       #return_sfc21 := FILL(BVAL := #fill_value_0, BLK    =>  "CTL");
       #return_sfc21 := FILL(BVAL := #fill_value_0, BLK    =>  "CRUC");
       #return_sfc21 := FILL(BVAL := #fill_value_0, BLK    =>  "CM_SEL_CTRL_ALG_DB");
       #return_sfc21 := FILL(BVAL := #fill_value_0, BLK    =>  "AM_BY2_RP_CALC_INC_DB");
       #return_sfc21 := FILL(BVAL := #fill_value_0, BLK    =>  "AM_PRS_CTRL_DB");
       #return_sfc21 := FILL(BVAL := #fill_value_0, BLK    =>  "AM_XT_DRV_MOVE_DB");
       #return_sfc21 := FILL(BVAL := #fill_value_0, BLK    =>  "AM_CR_DRV_MOVE_DB");
       #return_sfc21 := FILL(BVAL := #fill_value_0, BLK    =>  "AM_CTRL_DB");
       #return_sfc21 := FILL(BVAL := #fill_value_0, BLK    =>  "AM_ID_DB");
       #return_sfc21 := FILL(BVAL := #fill_value_0, BLK    =>  "AM_PD_DB");
       #return_sfc21 := FILL(BVAL := #fill_value_0, BLK    =>  "AM_ME_DB");
       #return_sfc21 := FILL(BVAL := #fill_value_0, BLK    =>  "AM_DI_DB");
       #return_sfc21 := FILL(BVAL := #fill_value_0, BLK    =>  "AM_NE_DB");
       #return_sfc21 := FILL(BVAL := #fill_value_0, BLK    =>  "AM_SH_DB");
       #return_sfc21 := FILL(BVAL := #fill_value_0, BLK    =>  "AM_BY_DB");
       #return_sfc21 := FILL(BVAL := #fill_value_0, BLK    =>  "AM_EC_DB");
       #return_sfc21 := FILL(BVAL := #fill_value_0, BLK    =>  "AM_SD_DB");
       #return_sfc21 := FILL(BVAL := #fill_value_0, BLK    =>  "AM_RE_DB");
       #return_sfc21 := FILL(BVAL := #fill_value_0, BLK    =>  "AM_EMG_DB");
       #return_sfc21 := FILL(BVAL := #fill_value_0, BLK    =>  "BM_CALL_DRV_DB");
       #return_sfc21 := FILL(BVAL := #fill_value_0, BLK    =>  "BM_CALL_HTR_CTRL_DB");
       #return_sfc21 := FILL(BVAL := #fill_value_0, BLK    =>  "BM_CALL_RES_CALC_DB");
       #return_sfc21 := FILL(BVAL := #fill_value_0, BLK    =>  "BM_MCC_DB");
       //return_sfc21 := FILL_SFC21(bval := fill_value_0, blk    :=  BM_XT_WGT_CALC_DB);
       //return_sfc21 := FILL_SFC21(bval := fill_value_0, blk    :=  BM_ROT_DRV_DIR_DB);
       //return_sfc21 := FILL_SFC21(bval := fill_value_0, blk    :=  BM_OP_CALL_DB);
       //return_sfc21 := FILL_SFC21(bval := fill_value_0, blk    :=  BM_FDR_MOVE_HOME_DB);
       //return_sfc21 := FILL_SFC21(bval := fill_value_0, blk    :=  BM_FDR_SEQ_DB);
       //return_sfc21 := FILL_SFC21(bval := fill_value_0, blk    :=  BM_FDR_LEAK_TST_DB);
       #return_sfc21 := FILL(BVAL := #fill_value_0, BLK    =>  "BM_SI_FIL_REG_DB");
       //return_sfc21 := FILL_SFC21(bval := fill_value_0, blk    :=  BM_XT_ORB_DET_DB);
       #return_sfc21 := FILL(BVAL := #fill_value_0, BLK    =>  "BM_MLT_LVL_MON_DB");
       //return_sfc21 := FILL_SFC21(bval := fill_value_0, blk    :=  BM_MLT_VIB_MON_DB);
       #return_sfc21 := FILL(BVAL := #fill_value_0, BLK    =>  "BM_ACC_MAIN_DB");
END_FUNCTION

FUNCTION "CM_CYCLE_RAMP" : Void   // FC320, SCL
{ S7_Optimized_Access := 'FALSE' }
VERSION : 0.0
// --------------------------------------------------------------------------------
//     program     :    CM_CYCLE_RAMP
//     description :    ramp function, called in cycle with timeflag  
//     name        :    hp
//     date        :    04.04.2000
// 
//     revision    :    
//     name        :    
//     date        :    
// 
//                     (c)CGS
//     --------------------------------------------------------------------------------
   VAR_INPUT
      SetpVal : Real;   // setpoint
      IncVal : Real;   // increment/decrement - value
      TimeFlag : Bool;   // time control flag
      Enable : Bool;   // Ramp enable / disable
   END_VAR
   VAR_IN_OUT
      ActVal : Real;   // actual value - input/output
   END_VAR
   VAR_TEMP
      act : Real;
   END_VAR
BEGIN


   IF #Enable THEN          //** Ramp function **

       #act := #ActVal;

       IF #TimeFlag THEN                // calculation only if true

           IF #SetpVal > #act THEN
               #act := #act + #IncVal;
               IF #act > #SetpVal THEN
                   #act := #SetpVal;
               END_IF;        
           ELSE
               IF #SetpVal < #act THEN
                   #act := #act - #IncVal;
                   IF #act < #SetpVal THEN
                       #act := #SetpVal;
                   END_IF;            
               ELSE
                   #act := #SetpVal;
               END_IF;
           END_IF;

       END_IF;

       #ActVal := #act;

   ELSE                //** no ramp function **

       #ActVal := #SetpVal;

   END_IF;
END_FUNCTION

FUNCTION "PM_HAI_CONVERT" : Real   // FC400, SCL
{ S7_Optimized_Access := 'FALSE' }
VERSION : 0.0
// --------------------------------------------------------------------------------
//     program     :    PM_HAI_CONVERT
//     description :    fetch, convert and scale  analog input signal       
//     name        :    hp
//     date        :    06.09.00
// 
//     revision    :    
//     name        :    
//     date        :    
//     
// 
//                     (c)CGS
//     --------------------------------------------------------------------------------
// hardware_type  min_value    max_value    function
//      1         0            +27648       linear    (0..10 V or 0..20 mA) Siemens
//      2         -27648       +27648       linear    (+/-10 V)
//      3         0            +32766       linear    (0..10 V or 0..20 mA) Beckhoff
//      4         -32767       +32766       linear    (+/-10 V)
   VAR_INPUT
      CHANNEL : Word;
      CONVERT_PAR : Struct
         hardware_type : Int;
         convert_type : Int;
         min_value : Real;
         max_value : Real;
      END_STRUCT;
   END_VAR
   VAR_TEMP
      input_real : Real;
      max_range : Real;
      min_range : Real;
   END_VAR
BEGIN


       #input_real := INT_TO_REAL (WORD_TO_INT (#CHANNEL));               //fetch input

       IF #CONVERT_PAR.hardware_type = 1 THEN                             // ao_type 1 [0..27648/lin] 

           #max_range := 27648;                                          //input limits 
           #min_range := 0;
           IF #input_real > #max_range THEN
               #input_real := #max_range; 
           END_IF;
           IF #input_real < #min_range THEN
               #input_real := #min_range; 
           END_IF;
                                                                        //calculate input value 
           //calculate input value 
           #input_real := #input_real/#max_range;   

           //set return value
           #PM_HAI_CONVERT := #input_real;

       END_IF;


       IF #CONVERT_PAR.hardware_type = 2 THEN                             // ao_type 2 [-27648..27648/lin] 

           #max_range := 27648;                                          //input limits 
           #min_range := -27648;
           IF #input_real > #max_range THEN
               #input_real := #max_range; 
           END_IF;
           IF #input_real < #min_range THEN
               #input_real := #min_range; 
           END_IF;

           //calculate input value 
           #input_real := #input_real/#max_range;   

           //set return value
        #PM_HAI_CONVERT := #input_real;

       END_IF;


       IF #CONVERT_PAR.hardware_type = 3 THEN                         // ai_type 3 [0..32766/lin]

           #max_range := 32766;                                      //input limits 
           #min_range := 0;

           IF #input_real > #max_range THEN
               #input_real := #max_range; 
           END_IF;
           IF #input_real < #min_range THEN
               #input_real := #min_range; 
           END_IF;


           //calculate input value 
           #input_real := #input_real/#max_range; 

           //set return value
           #PM_HAI_CONVERT := #input_real;

       END_IF;


       IF #CONVERT_PAR.hardware_type = 4 THEN                  // ai_type 4 [-32767..32766/lin] 

           #max_range := 32766;                               //input limits 
           #min_range := -32767;
           IF #input_real > #max_range THEN
               #input_real := #max_range; 
           END_IF;
           IF #input_real < #min_range THEN
               #input_real := #min_range; 
           END_IF;

           //calculate input value 
           #input_real := #input_real/#max_range; 

           //set return value
           #PM_HAI_CONVERT := #input_real;

       END_IF;
END_FUNCTION

FUNCTION "PM_HAO_CONVERT" : Word   // FC401, SCL
{ S7_Optimized_Access := 'FALSE' }
VERSION : 0.0
// --------------------------------------------------------------------------------
//     program     :    PM_HAO_CONVERT
//     description :    convert, scale and write analog output signal       
//     name        :    hp
//     date        :    06.09.00
//     
//     revision    :
//     name        :
//     date        :    
//                     (c)CGS
//     --------------------------------------------------------------------------------
// hardware_type  min_value    max_value    function    
//      1         0            +27648       linear    (0..10 V or 0..20 mA)    Siemens
//      2         -27648       +27648       linear    (+/- 10 V)      
//      3         0            +32766       linear    (0..10 V or 0..20 mA)    Beckhoff
//      4         -32767       +32766       linear     (+/- 10V)
   VAR_INPUT
      OUTVALUE : Real;
      CONVERT_PAR : Struct
         hardware_type : Int;
         convert_type : Int;
         min_value : Real;
         max_value : Real;
      END_STRUCT;
   END_VAR
   VAR_TEMP
      output_real : Real;
      max_range : Real;
      min_range : Real;
   END_VAR
BEGIN


       #output_real := #OUTVALUE;                                        //fetch output value

       IF #output_real > 1.0 THEN                                          //upper input limits
           #output_real := 1.0; 
       END_IF;


       IF #CONVERT_PAR.hardware_type = 1 THEN                            // ao_type 1 [0..27648/lin] 

           IF #output_real < 0.0 THEN                                     //set lower limit
               #output_real := 0.0; 
           END_IF;

           #max_range := 27648;                                          //set output range                                  
           #min_range := 0;

           //calculate output value 
           #output_real := #output_real*#max_range;   

       END_IF;

       IF #CONVERT_PAR.hardware_type = 2 THEN                             // ao_type 2 [-27648..27648/lin] 

           IF #output_real < -1.0 THEN                                     //set lower limit
               #output_real := -1.0; 
           END_IF;

           #max_range := 27648;                                          //set output range 
           #min_range := -27648;

           //calculate output value
           #output_real := #output_real*#max_range;   

       END_IF;

       IF #CONVERT_PAR.hardware_type = 3 THEN                             // ao_type 3 [0..32766/lin] 

           IF #output_real < 0.0 THEN                                     //set lower limit
               #output_real := 0.0; 
           END_IF;

           #max_range := 32766;                                          //set output range 
           #min_range := 0;

           //calculate output value
           #output_real := #output_real*#max_range;   

       END_IF;

       IF #CONVERT_PAR.hardware_type = 4 THEN                             // ao_type 4 [-32767..32766/lin] 

           IF #output_real < -1.0 THEN                                    //set lower limit
               #output_real := -1.0; 
           END_IF;

           #max_range := 32766;                                         //set output range 
           #min_range := -32767;

           //calculate output value
           #output_real := #output_real*#max_range;   

       END_IF;

   #PM_HAO_CONVERT := INT_TO_WORD(REAL_TO_INT(#output_real));                //set return value                                           //set return value
END_FUNCTION

FUNCTION "PM_HAI" : Void   // FC402, SCL
{ S7_Optimized_Access := 'FALSE' }
VERSION : 0.0
// --------------------------------------------------------------------------------
//     program:         PM_HAI
//     description :    automatically generated PM_HAI
//     name:            hp
//     date        :    03.02.2021
// 
//     revision:
//     name:
//     Date:
//                     (c)CGS
//     --------------------------------------------------------------------------------
   VAR_TEMP
      x : Bool;
   END_VAR
BEGIN


   IF NOT "SY".SIM_ON THEN

       "HAI".TRV_ACT_POS := "PM_HAI_CONVERT" (CHANNEL := "P_HAI_TRV_ACT_POS":P, CONVERT_PAR := "CAI".CONFIG_DATA[1]);
       "HAI".TRV_ACT_POS_1 := "PM_HAI_CONVERT" (CHANNEL := "P_HAI_TRV_ACT_POS_1":P, CONVERT_PAR := "CAI".CONFIG_DATA[2]);
       "HAI".TRV_PRS_FIL_1 := "PM_HAI_CONVERT" (CHANNEL := "P_HAI_TRV_PRS_FIL_1":P, CONVERT_PAR := "CAI".CONFIG_DATA[3]);
       "HAI".TRV_PRS_FIL_2 := "PM_HAI_CONVERT" (CHANNEL := "P_HAI_TRV_PRS_FIL_2":P, CONVERT_PAR := "CAI".CONFIG_DATA[4]);
       "HAI".PYR_ACT_HTR_1_TMP := "PM_HAI_CONVERT" (CHANNEL := "P_HAI_PYR_ACT_HTR_1_TMP":P, CONVERT_PAR := "CAI".CONFIG_DATA[5]);
       "HAI".ACT_PRS_AR_VSL := "PM_HAI_CONVERT" (CHANNEL := "P_HAI_ACT_PRS_AR_VSL":P, CONVERT_PAR := "CAI".CONFIG_DATA[6]);
       "HAI".PYR_ACT_MELT_TMP := "PM_HAI_CONVERT" (CHANNEL := "P_HAI_PYR_ACT_MELT_TMP":P, CONVERT_PAR := "CAI".CONFIG_DATA[7]);
       "HAI".GCH_PCR_ACT_PRS := "PM_HAI_CONVERT" (CHANNEL := "P_HAI_GCH_PCR_ACT_PRS":P, CONVERT_PAR := "CAI".CONFIG_DATA[8]);
       "HAI".FCH_PCR_ACT_PRS := "PM_HAI_CONVERT" (CHANNEL := "P_HAI_FCH_PCR_ACT_PRS":P, CONVERT_PAR := "CAI".CONFIG_DATA[9]);
       "HAI".FCH_BAR_ACT_PRS_100 := "PM_HAI_CONVERT" (CHANNEL := "P_HAI_FCH_BAR_ACT_PRS_100":P, CONVERT_PAR := "CAI".CONFIG_DATA[10]);
       "HAI".ACC_WTR_TMP := "PM_HAI_CONVERT" (CHANNEL := "P_HAI_ACC_WTR_TMP":P, CONVERT_PAR := "CAI".CONFIG_DATA[11]);
       "HAI".ACC_WTR_PRS_IN := "PM_HAI_CONVERT" (CHANNEL := "P_HAI_ACC_WTR_PRS_IN":P, CONVERT_PAR := "CAI".CONFIG_DATA[12]);
       "HAI".ACC_WTR_FLW_OUT := "PM_HAI_CONVERT" (CHANNEL := "P_HAI_ACC_WTR_FLW_OUT":P, CONVERT_PAR := "CAI".CONFIG_DATA[13]);
       "HAI".ACC_WTR_FLW_IN := "PM_HAI_CONVERT" (CHANNEL := "P_HAI_ACC_WTR_FLW_IN":P, CONVERT_PAR := "CAI".CONFIG_DATA[14]);
       "HAI".ACC_WTR_SPL_PRS := "PM_HAI_CONVERT" (CHANNEL := "P_HAI_ACC_WTR_SPL_PRS":P, CONVERT_PAR := "CAI".CONFIG_DATA[15]);
       "HAI".ACC_SPARE_810 := "PM_HAI_CONVERT" (CHANNEL := "P_HAI_ACC_SPARE_810":P, CONVERT_PAR := "CAI".CONFIG_DATA[16]);

   END_IF;
END_FUNCTION

FUNCTION "PM_HAO" : Void   // FC403, SCL
{ S7_Optimized_Access := 'FALSE' }
VERSION : 0.0
// --------------------------------------------------------------------------------
//     program:         PM_HAO
//     description :    automatically generated PM_HAO
//     name:            hp
//     date        :    03.02.2021
// 
//     revision:
//     name:
//     Date:
//                     (c)CGS
//     --------------------------------------------------------------------------------
   VAR_TEMP
      x : Bool;
   END_VAR
BEGIN


   IF NOT "SY".SIM_ON THEN

       "P_HAO_TRV_SET_POS":P := "PM_HAO_CONVERT"(OUTVALUE := "HAO".TRV_SET_POS, CONVERT_PAR := "CAO".CONFIG_DATA[1]);
       "P_HAO_TRV_SET_POS_1":P := "PM_HAO_CONVERT"(OUTVALUE := "HAO".TRV_SET_POS_1, CONVERT_PAR := "CAO".CONFIG_DATA[2]);

   END_IF;
END_FUNCTION

FUNCTION "BM_SET_DIS_VAR" : Void   // FC503, SCL
{ S7_Optimized_Access := 'FALSE' }
VERSION : 0.0
BEGIN


       //heater 2
       //--------
       "DIS".ACT_HTR_2_AV_TMP := "AV".AVG_HTR_2_TMP;            //set display values
       "DIS".ACT_HTR_2_TMP := "AV".ACT_HTR_2_TMP;

       //pressure and gas flow
       //---------------------
       "DIS".SET_PRS_FNC   := "KYA".SET_PRS_FNC;

       "DIS".SET_GAS_1_FLW := "KYA".SET_GAS_1_FLW;
       "DIS".SET_GAS_2_FLW := "KYA".SET_GAS_2_FLW;

       "DIS".ACT_CR_POS_DIPPING    := "KYA".SET_DIP_POS_CR;
       "DIS".ACT_BDY2_LEN          := "KYA".ACT_BDY2_LEN;

       //melt contact variable copied to logging variable
       //------------------------------------------------
       "DIS".XT_MELT_CONTACT :=  INT_TO_REAL(BOOL_TO_INT("LT".XT_MELT_CONTACT));

       //Presetting after PLC restart
       //----------------------------
       IF ("SY".RUN_TIME < 5)  THEN
           "KYA".SET_XT_LFT_GN   := 1.0;     // gain values for drive calibration EKZ 2700 (old hardware)
           "KYA".SET_XT_ROT_GN   := 1.0;
           "KYA".SET_CR_LFT_GN   := 1.0;
           "KYA".SET_CR_ROT_GN   := 1.0;

           "KYA".SET_THR_CAL_FACT    := 1.0; // threshold calibration factor
       END_IF;
END_FUNCTION

ORGANIZATION_BLOCK "MAIN_OB1"   // OB1, SCL
{ S7_Optimized_Access := 'FALSE' }
VERSION : 0.0
// --------------------------------------------------------------------------------
//     program     :    MAIN_OB1
//     description :    main program scan OB1        
//     name        :    K. Kalkowski
//     date        :    01.09.99
// 
//     revision    :    AM_CALL
//     name        :    D.Bruess
//     date        :    23.11.99
//                     
//                     (c)CGS                    
//     --------------------------------------------------------------------------------
   VAR_TEMP
      OB1_EV_CLASS : Byte;   // Bits 0-3 = 1 (Coming event), Bits 4-7 = 1 (Event class 1)
      OB1_SCAN_1 : Byte;   // 1 (Cold restart scan 1 of OB 1), 3 (Scan 2-n of OB 1)
      OB1_PRIORITY : Byte;   // Priority of OB Execution
      OB1_OB_NUMBR : Byte;   // 1 (Organization block 1, OB1)
      OB1_RESERVED_1 : Byte;   // Reserved for system
      OB1_RESERVED_2 : Byte;   // Reserved for system
      OB1_PREV_CYCLE : Int;   // Cycle time of previous OB1 scan (milliseconds)
      OB1_MIN_CYCLE : Int;   // Minimum cycle time of OB1 (milliseconds)
      OB1_MAX_CYCLE : Int;   // Maximum cycle time of OB1 (milliseconds)
      OB1_DATE_TIME : Date_And_Time;   // Date and time OB1 started
   END_VAR
BEGIN

       //write cycle information
       //-----------------------
       "SY".OB1_PREV_CYCLE   :=  #OB1_PREV_CYCLE;         //Cycle time of previous OB1 scan (milliseconds)
       "SY".OB1_MIN_CYCLE    :=  #OB1_MIN_CYCLE;          //Minimum cycle time of OB1 (milliseconds)
       "SY".OB1_MAX_CYCLE    :=  #OB1_MAX_CYCLE;          //Maximum cycle time of OB1 (milliseconds)


       //call global DP diagnosis
       //------------------------
       "PM_PN_SET_FLT_MSG"();
       "CALL_PN_DIAG"();     

       //call power fail control
       //-----------------------  
      // SM_PWR_FAIL.SM_PWR_FAIL_DB();

       //ACTUAL PLC VERSION AND CONFIGURATION
       //------------------------------------
       "DIS".ACT_PLC_VERSION := "SW".ACT_PLC_VERSION;
       "DIS".ACT_PLC_CONFIG  := "SW".ACT_PLC_CONFIG;       

       //Build alarm acknowledge for one cycle
       //-------------------------------------
       "DV".ALARM_ACKN       := "KYD".ALARM_ACKN AND NOT "DV".ALARM_ACKN_OLD;
       "DV".ALARM_ACKN_OLD   := "KYD".ALARM_ACKN;

       //System Time
       //-----------
       "SysTimeFlag"();

       "PM_CALL_ST"();
       "BM_CALL"();

       //calculate crucible geometry
       // --------------------------
       "CM_CRUC_MAIN"();

       //automatic sequence
       // -----------------
       "AM_CTRL_DB"();

       //alarm management
       //----------------
       "SM_FLT_SETP_DEV_PRC_DB"();
       "SM_FLT_SET_ALM"();
       "SM_CALL_FAULT_RESET"();
END_ORGANIZATION_BLOCK

ORGANIZATION_BLOCK "ITR_1000ms_OB32"   // OB32, SCL
{ S7_Optimized_Access := 'FALSE' }
VERSION : 0.0
// --------------------------------------------------------------------------------
//     program     :    ITR_1000ms_OB32
//     description :    cyclic interrupt OB32 1000ms        
//     name        :    G. Eibelsh鋟ser
//     date        :    01.09.99
// 
//     revision    :
//     name        :
//     date        :    
//                     (c)CGS
//     --------------------------------------------------------------------------------
   VAR_TEMP
      info : Array[0..19] of Byte;
   END_VAR
BEGIN

       "SY".RUN_TIME := "SY".RUN_TIME + 1;             //count time since last reset
       "AM_TIME"();                                  //call timer function
       "BM_CALL_RES_CALC_DB"();     //calculate heater resistance
END_ORGANIZATION_BLOCK

ORGANIZATION_BLOCK "ITR_100ms_OB35"   // OB35, SCL
{ S7_Optimized_Access := 'FALSE' }
VERSION : 0.0
// --------------------------------------------------------------------------------
//     program     :    ITR_100ms_OB35
//     description :    cyclic interrupt OB35 100ms        
//     name        :    K. Kalkowski
//     date        :    01.09.99
// 
//     revision    :
//     name        :
//     date        :    
//                     (c)CGS
//     --------------------------------------------------------------------------------
   VAR_TEMP
      info : Array[0..19] of Byte;
   END_VAR
BEGIN

       "CM_CALL_100MS"();                               //call control loop modules

       IF "APC".STATUS="APC".BODY AND "APC".BYRST THEN
           "AM_BY2_RP_CALC_INC_DB"();    //call increment calc.fnc for 2nd body ramp

       END_IF;
END_ORGANIZATION_BLOCK

ORGANIZATION_BLOCK "ERR_TIME_OB80"   // OB80, SCL
{ S7_Optimized_Access := 'FALSE' }
VERSION : 0.0
// --------------------------------------------------------------------------------
//     program     :    ERR_TIME_OB80
//     description :    time error OB80        
//     name        :    K. Kalkowski
//     date        :    01.09.99
// 
//     revision    :
//     name        :
//     date        :    
//                     (c)CGS
//     --------------------------------------------------------------------------------
   VAR_TEMP
      info : Array[0..19] of Byte;
   END_VAR
BEGIN

       ;
END_ORGANIZATION_BLOCK

ORGANIZATION_BLOCK "ITR_DIAGNOSTIC_OB82"   // OB82, SCL
{ S7_Optimized_Access := 'FALSE' }
VERSION : 0.0
// --------------------------------------------------------------------------------
//     program     :    ITR_DIAGNOSTIC_OB82
//     description :    diagnostic interrupt OB82     
//     name        :    G. Eibelsh鋟ser
//     date        :    01.09.99
// 
//     revision    :
//     name        :
//     date        :    
//                     (c)CGS
//     --------------------------------------------------------------------------------
   VAR_TEMP
      info : Array[0..19] of Byte;
   END_VAR
BEGIN

    ;
END_ORGANIZATION_BLOCK

ORGANIZATION_BLOCK "ITR_MODULE_OB83"   // OB83, SCL
{ S7_Optimized_Access := 'FALSE' }
VERSION : 0.0
// --------------------------------------------------------------------------------
//     program     :    ITR_MODULE_OB83
//     description :    insert/remove module interrupt OB83 <NOT USED!>       
//     name        :    K. Kalkowski
//     date        :    01.09.99
// 
//     revision    :
//     name        :
//     date        :    
//                     (c)CGS
//     --------------------------------------------------------------------------------
   VAR_TEMP
      info : Array[0..19] of Byte;
   END_VAR
BEGIN

       ;
END_ORGANIZATION_BLOCK

ORGANIZATION_BLOCK "ERR_PRI_CLASS_OB85"   // OB85, SCL
{ S7_Optimized_Access := 'FALSE' }
VERSION : 0.0
// --------------------------------------------------------------------------------
//     program     :    ERR_PRI_CLASS_OB85
//     description :    priority class error OB85         
//     name        :    K. Kalkowski
//     date        :    01.09.99
// 
//     revision    :
//     name        :
//     date        :    
//                     (c)CGS
//     --------------------------------------------------------------------------------
   VAR_TEMP
      info : Array[0..19] of Byte;
   END_VAR
BEGIN

       ;
END_ORGANIZATION_BLOCK

ORGANIZATION_BLOCK "ERR_RACK_OB86"   // OB86, SCL
{ S7_Optimized_Access := 'FALSE' }
VERSION : 0.0
// --------------------------------------------------------------------------------
//     program     :    ERR_RACK_OB86
//     description :    rack failure OB86         
//     name        :    G. Eibelsh鋟ser
//     date        :    01.09.99
// 
//     revision    :
//     name        :
//     date        :    
//                     (c)CGS
//     --------------------------------------------------------------------------------
   VAR_TEMP
      info : Array[0..19] of Byte;
   END_VAR
BEGIN

      ;
END_ORGANIZATION_BLOCK

ORGANIZATION_BLOCK "RESET_OB100"   // OB100, SCL
{ S7_Optimized_Access := 'FALSE' }
VERSION : 0.0
// --------------------------------------------------------------------------------
//     program     :    RESET_OB100
//     description :    cold restart OB100         
//     name        :    K. Kalkowski
//     date        :    01.09.99
// 
//     revision    :
//     name        :
//     date        :    
//                     (c)CGS
//     --------------------------------------------------------------------------------
   VAR_TEMP
      info : Array[0..19] of Byte;
   END_VAR
BEGIN

       "SM_RESTART_CALL"();
   ;
END_ORGANIZATION_BLOCK

ORGANIZATION_BLOCK "ERR_PROG_OB121"   // OB121, SCL
{ S7_Optimized_Access := 'FALSE' }
VERSION : 0.0
// --------------------------------------------------------------------------------
//     program     :    ERR_PROG_OB121
//     description :    programming error OB121         
//     name        :    K. Kalkowski
//     date        :    01.09.99
// 
//     revision    :
//     name        :
//     date        :    
//                     (c)CGS
//     --------------------------------------------------------------------------------
   VAR_TEMP
      info : Array[0..19] of Byte;
   END_VAR
BEGIN

       ;
END_ORGANIZATION_BLOCK

ORGANIZATION_BLOCK "ERR_ACCESS_OB122"   // OB122, SCL
{ S7_Optimized_Access := 'FALSE' }
VERSION : 0.0
// --------------------------------------------------------------------------------
//     program     :    ERR_ACCESS_OB122
//     description :    access error OB122        
//     name        :    K. Kalkowski
//     date        :    01.09.99
// 
//     revision    :
//     name        :
//     date        :    
//                     (c)CGS
//     --------------------------------------------------------------------------------
   VAR_TEMP
      info : Array[0..19] of Byte;
   END_VAR
BEGIN

       ;
END_ORGANIZATION_BLOCK

// ===== PLC "CPU 315-2 PN/DP"  Unspecific CPU S7 300 =====
// protected blocks, not shown: "ERR_ACCESS_OB122", "ERR_PRI_CLASS_OB85", "ERR_PROG_OB121", "ERR_RACK_OB86", "ERR_TIME_OB80", "IO_LINK_MASTER", "ITR_1000ms_OB32", "ITR_100ms_OB35", "ITR_DIAGNOSTIC_OB82", "RESET_OB100"

VAR_GLOBAL   // PLC tag table "STEP7 classic symbols"
   "Tag_1" AT %ED1028 : DWord;
   "Tag_2" AT %AD256 : DWord;
   "Tag_3" AT %EB1032 : Byte;
   "Tag_4" AT %AB260 : Byte;
   "Tag_5" AT %ED1037 : DWord;
   "Tag_6" AT %AD262 : DWord;
   "Tag_7" AT %EB1041 : Byte;
   "Tag_8" AT %AB266 : Byte;
   "Tag_9" AT %ED1046 : DWord;
   "Tag_10" AT %AD268 : DWord;
   "Tag_11" AT %EB1050 : Byte;
   "Tag_12" AT %AB272 : Byte;
   "Tag_13" AT %ED1055 : DWord;
   "Tag_14" AT %AD274 : DWord;
   "Tag_15" AT %EB1059 : Byte;
   "Tag_16" AT %AB278 : Byte;
   "Tag_17" AT %ED1064 : DWord;
   "Tag_18" AT %AD280 : DWord;
   "Tag_19" AT %EB1068 : Byte;
   "Tag_20" AT %AB284 : Byte;
   "Tag_21" AT %ED1073 : DWord;
   "Tag_22" AT %AD286 : DWord;
   "Tag_23" AT %EB1077 : Byte;
   "Tag_24" AT %AB290 : Byte;
   "Tag_25" AT %ED1100 : DWord;
   "Tag_26" AT %AD304 : DWord;
   "Tag_27" AT %EB1104 : Byte;
   "Tag_28" AT %AB308 : Byte;
   "Tag_29" AT %ED1109 : DWord;
   "Tag_30" AT %AD310 : DWord;
   "Tag_31" AT %EB1113 : Byte;
   "Tag_32" AT %AB314 : Byte;
   "Tag_33" AT %ED1118 : DWord;
   "Tag_34" AT %AD316 : DWord;
   "Tag_35" AT %EB1122 : Byte;
   "Tag_36" AT %AB320 : Byte;
   "Tag_37" AT %ED1127 : DWord;
   "Tag_38" AT %AD322 : DWord;
   "Tag_39" AT %EB1131 : Byte;
   "Tag_40" AT %AB326 : Byte;
   "Tag_41" AT %ED1136 : DWord;
   "Tag_42" AT %AD328 : DWord;
   "Tag_43" AT %EB1140 : Byte;
   "Tag_44" AT %AB332 : Byte;
   "Tag_45" AT %ED1172 : DWord;
   "Tag_46" AT %AD352 : DWord;
   "Tag_47" AT %EB1176 : Byte;
   "Tag_48" AT %AB356 : Byte;
   "Tag_49" AT %ED1181 : DWord;
   "Tag_50" AT %AD358 : DWord;
   "Tag_51" AT %EB1185 : Byte;
   "Tag_52" AT %AB362 : Byte;
   "Tag_53" AT %ED1190 : DWord;
   "Tag_54" AT %AD364 : DWord;
   "Tag_55" AT %EB1194 : Byte;
   "Tag_56" AT %AB368 : Byte;
   "Tag_57" AT %ED1199 : DWord;
   "Tag_58" AT %AD370 : DWord;
   "Tag_59" AT %EB1203 : Byte;
   "Tag_60" AT %AB374 : Byte;
   "Tag_61" AT %ED1208 : DWord;
   "Tag_62" AT %AD376 : DWord;
   "Tag_63" AT %EB1212 : Byte;
   "Tag_64" AT %AB380 : Byte;
   "Tag_65" AT %ED1217 : DWord;
   "Tag_66" AT %AD382 : DWord;
   "Tag_67" AT %EB1221 : Byte;
   "Tag_68" AT %AB386 : Byte;
   "Tag_69" AT %ED1226 : DWord;
   "Tag_70" AT %AD388 : DWord;
   "Tag_71" AT %EB1230 : Byte;
   "Tag_72" AT %AB392 : Byte;
   "Tag_73" AT %ED1244 : DWord;
   "Tag_74" AT %AD400 : DWord;
   "Tag_75" AT %EB1248 : Byte;
   "Tag_76" AT %AB404 : Byte;
   "Tag_77" AT %ED1253 : DWord;
   "Tag_78" AT %AD406 : DWord;
   "Tag_79" AT %EB1257 : Byte;
   "Tag_80" AT %AB410 : Byte;
   "Tag_81" AT %ED1262 : DWord;
   "Tag_82" AT %AD412 : DWord;
   "Tag_83" AT %EB1266 : Byte;
   "Tag_84" AT %AB416 : Byte;
   "Tag_85" AT %ED1271 : DWord;
   "Tag_86" AT %AD418 : DWord;
   "Tag_87" AT %EB1275 : Byte;
   "Tag_88" AT %AB422 : Byte;
   "Tag_89" AT %ED1280 : DWord;
   "Tag_90" AT %AD424 : DWord;
   "Tag_91" AT %EB1284 : Byte;
   "Tag_92" AT %AB428 : Byte;
   "Tag_93" AT %ED1289 : DWord;
   "Tag_94" AT %AD430 : DWord;
   "Tag_95" AT %EB1293 : Byte;
   "Tag_96" AT %AB434 : Byte;
END_VAR

ORGANIZATION_BLOCK "MAIN_OB1"   // OB1, STL
TITLE = "Main Program Sweep (Cycle)"
{ S7_Optimized_Access := 'FALSE' }
VERSION : 0.1
// ifm io-link master Adresse transport
   VAR_TEMP
      OB1_EV_CLASS : Byte;   // Bits 0-3 = 1 (Coming event), Bits 4-7 = 1 (Event class 1)
      OB1_SCAN_1 : Byte;   // 1 (Cold restart scan 1 of OB 1), 3 (Scan 2-n of OB 1)
      OB1_PRIORITY : Byte;   // Priority of OB Execution
      OB1_OB_NUMBR : Byte;   // 1 (Organization block 1, OB1)
      OB1_RESERVED_1 : Byte;   // Reserved for system
      OB1_RESERVED_2 : Byte;   // Reserved for system
      OB1_PREV_CYCLE : Int;   // Cycle time of previous OB1 scan (milliseconds)
      OB1_MIN_CYCLE : Int;   // Minimum cycle time of OB1 (milliseconds)
      OB1_MAX_CYCLE : Int;   // Maximum cycle time of OB1 (milliseconds)
      OB1_DATE_TIME : Date_And_Time;   // Date and time OB1 started
   END_VAR
BEGIN

REGION Network 1

   //-------------------  crucible shaft
         L     "Tag_1":P;  // masse flow and temperature 4 Bytes transfer to I-Device
         T     "Tag_2":P;

         L     "Tag_3":P;  // PQI Status 2 Bytes transfer to I-Device
         T     "Tag_4":P;

   //-------------------- High current cable heater 1
         L     "Tag_5":P;
         T     "Tag_6":P;

         L     "Tag_7":P;
         T     "Tag_8":P;

   //-------------------- High current cable heater 2
         L     "Tag_9":P;
         T     "Tag_10":P;

         L     "Tag_11":P;
         T     "Tag_12":P;

   //-------------------- seed shaft
         L     "Tag_13":P;
         T     "Tag_14":P;

         L     "Tag_15":P;
         T     "Tag_16":P;

   //-------------------- Power supply heater
         L     "Tag_17":P;
         T     "Tag_18":P;

         L     "Tag_19":P;
         T     "Tag_20":P;

   //-------------------- gate chamber
         L     "Tag_21":P;
         T     "Tag_22":P;

         L     "Tag_23":P;
         T     "Tag_24":P;
   //-------------------- spare
   //      L     PED 1082
   //      T     PAD  292

   //      L     PEW 1086
   //      T     PAW  296

   //-------------------- spare
   //      L     PED 1091
   //      T     PAD  298

   //      L     PEW 1095
   //      T     PAW  302

   //-------------------- gate valve housing
         L     "Tag_25":P;
         T     "Tag_26":P;

         L     "Tag_27":P;
         T     "Tag_28":P;

   //-------------------- gate valve
         L     "Tag_29":P;
         T     "Tag_30":P;

         L     "Tag_31":P;
         T     "Tag_32":P;
   //-------------------- view port
         L     "Tag_33":P;
         T     "Tag_34":P;

         L     "Tag_35":P;
         T     "Tag_36":P;

   //-------------------- Gate chamber- view ports and bellow
         L     "Tag_37":P;
         T     "Tag_38":P;

         L     "Tag_39":P;
         T     "Tag_40":P;

   //-------------------- top chamber
         L     "Tag_41":P;
         T     "Tag_42":P;

         L     "Tag_43":P;
         T     "Tag_44":P;

   //-------------------- spare
   //     L     PED 1145
   //      T     PAD  334

   //      L     PEW 1149
   //      T     PAW  338

   //-------------------- spare
   //      L     PED 1154
   //      T     PAD  340

   //      L     PEW 1158
   //      T     PAW  344

   //-------------------- spare
   //      L     PED 1163
   //      T     PAD  346

   //      L     PEW 1167
   //      T     PAW  350   *)

   //-------------------- technology flange
         L     "Tag_45":P;
         T     "Tag_46":P;

         L     "Tag_47":P;
         T     "Tag_48":P;
   //-------------------- magnet compressor unit 4

         L     "Tag_49":P;
         T     "Tag_50":P;

         L     "Tag_51":P;
         T     "Tag_52":P;

   //-------------------- magnet compressor unit 3
         L     "Tag_53":P;
         T     "Tag_54":P;

         L     "Tag_55":P;
         T     "Tag_56":P;

   //-------------------- upper furnace vessel
         L     "Tag_57":P;
         T     "Tag_58":P;

         L     "Tag_59":P;
         T     "Tag_60":P;

   //-------------------- magnet compressor unit 2
         L     "Tag_61":P;
         T     "Tag_62":P;

         L     "Tag_63":P;
         T     "Tag_64":P;
   //-------------------- lower furnace vessel

         L     "Tag_65":P;
         T     "Tag_66":P;

         L     "Tag_67":P;
         T     "Tag_68":P;
   //-------------------- magnet compressor unit 1

         L     "Tag_69":P;
         T     "Tag_70":P;

         L     "Tag_71":P;
         T     "Tag_72":P;
   //-------------------- spare

   //      L     PED 1235
   //      T     PAD  394

   //      L     PEW 1239
   //      T     PAW  398

   //-------------------- bottom chamber
         L     "Tag_73":P;
         T     "Tag_74":P;

         L     "Tag_75":P;
         T     "Tag_76":P;
   //-------------------- Power supply magnet

         L     "Tag_77":P;
         T     "Tag_78":P;

         L     "Tag_79":P;
         T     "Tag_80":P;

   //-------------------- Socket bottom chamber
         L     "Tag_81":P;
         T     "Tag_82":P;

         L     "Tag_83":P;
         T     "Tag_84":P;

   //-------------------- Current feed through heater 1
         L     "Tag_85":P;
         T     "Tag_86":P;

         L     "Tag_87":P;
         T     "Tag_88":P;

   //-------------------- Current feed through heater 2
         L     "Tag_89":P;
         T     "Tag_90":P;

         L     "Tag_91":P;
         T     "Tag_92":P;

   //-------------------- vacuum bypass tube
         L     "Tag_93":P;
         T     "Tag_94":P;

         L     "Tag_95":P;
         T     "Tag_96":P;

   //-------------------- spare
   //     L     PED 1298
   //     T     PAD  436

   //     L     PEB 1302
   //     T     PAB  440

   //-------------------- spare
   //     L     PED 1307
   //     T     PAD  442

   //     L     PEB 1311
   //     T     PAB  446
END_REGION
END_ORGANIZATION_BLOCK

ORGANIZATION_BLOCK "I/O_FLT2"   // OB83, STL
TITLE = "I/O Point Fault"
{ S7_Optimized_Access := 'FALSE' }
VERSION : 0.1
   VAR_TEMP
      OB83_EV_CLASS : Byte;   // 16#38/39, Event class 3, module inserted/removed (8/9)
      OB83_FLT_ID : Byte;   // 16#XX, Fault identifcation code
      OB83_PRIORITY : Byte;   // Priority of OB Execution
      OB83_OB_NUMBR : Byte;   // 83 (Organization block 83, OB83)
      OB83_RESERVED_1 : Byte;   // Reserved for system
      OB83_MDL_ID : Byte;   // Input module (01010100), Output module (01010101)
      OB83_MDL_ADDR : Word;   // Base address of module with point fault
      OB83_RACK_NUM : Int;   // Number of rack that has module with point fault
      OB83_MDL_TYPE : Word;   // Module type with point fault
      OB83_DATE_TIME : Date_And_Time;   // Date and time OB83 started
   END_VAR
BEGIN
END_ORGANIZATION_BLOCK

// ===== PLC "Mig_PVA_AWL"  Unspecific CPU S7 300 =====
// protected blocks, not shown: "AG_LRECV_LF", "AG_LSEND_LF", "AG_RECV", "AG_SEND", "DCO_ReadDriveParameter", "DCO_WriteDriveParameter", "GLOBAL_DP_DIAG", "IO_LINK_DEVICE", "IO_LINK_MASTER"

VAR_GLOBAL   // PLC tag table "Default tag table"
   "Tag_1" AT %M0.0 : Bool;
   "Tag_2" AT %M0.1 : Bool;
   "Tag_3" AT %M1.0 : Bool;
   "Tag_4" AT %M1.1 : Bool;
   "Tag_5" AT %M1.2 : Bool;
   "Tag_6" AT %M1.3 : Bool;
   "Tag_7" AT %M1.4 : Bool;
   "Tag_8" AT %M1.5 : Bool;
   "Tag_9" AT %M1.6 : Bool;
   "Tag_10" AT %M1.7 : Bool;
   "Tag_11" AT %M2.0 : Bool;
   "Tag_12" AT %M3.0 : Bool;
   "Tag_13" AT %M3.1 : Bool;
   "Tag_14" AT %M2.1 : Bool;
   "Tag_15" AT %M3.2 : Bool;
   "Tag_16" AT %M3.3 : Bool;
   "Tag_17" AT %M2.2 : Bool;
   "Tag_18" AT %M3.4 : Bool;
   "Tag_19" AT %M3.5 : Bool;
   "Tag_20" AT %M2.3 : Bool;
   "Tag_21" AT %M3.6 : Bool;
   "Tag_22" AT %M3.7 : Bool;
   "Tag_23" AT %M2.4 : Bool;
   "Tag_24" AT %M4.0 : Bool;
   "Tag_25" AT %M4.1 : Bool;
   "Tag_26" AT %M2.5 : Bool;
   "Tag_27" AT %M4.2 : Bool;
   "Tag_28" AT %M4.3 : Bool;
   "Tag_29" AT %M2.6 : Bool;
   "Tag_30" AT %M4.4 : Bool;
   "Tag_31" AT %M4.5 : Bool;
   "Tag_32" AT %M2.7 : Bool;
   "Tag_33" AT %M4.6 : Bool;
   "Tag_34" AT %M4.7 : Bool;
END_VAR

DATA_BLOCK "BM_GRW_REC_BOOL"   // DB701
{ S7_Optimized_Access := 'FALSE' }
VERSION : 0.0
// --------------------------------------------------------------------------------
// program:             GRW_REC_BOOL
// description :        bool data for growth record
// name:                mb
// date        :        27.11.09 
// --------------------------------------------------------------------------------
   VAR
      phase_restart : Bool;   // Phase wurde neu gestartet
      phase_spare_02 : Bool;
      phase_spare_03 : Bool;
      phase_spare_04 : Bool;
      phase_spare_05 : Bool;
      phase_spare_06 : Bool;
      phase_spare_07 : Bool;
      phase_spare_08 : Bool;
      phase_spare_09 : Bool;
      phase_spare_10 : Bool;   // pump down
      pd_min_prs_reached : Bool;   // min. Druck erreicht
      pd_failed : Bool;   // Leckrate (0=ok/1=nicht ok)
      pd_new_seed : Bool;   // neuer Impfling bei Prozesstart
      pd_spare_04 : Bool;
      pd_spare_05 : Bool;
      pd_spare_06 : Bool;
      pd_spare_07 : Bool;
      pd_spare_08 : Bool;
      pd_spare_09 : Bool;
      pd_spare_10 : Bool;   // melting
      me_completed : Bool;   // Einschmelzen beendet (von Kamera erkannt)
      me_spare_02 : Bool;
      me_spare_03 : Bool;
      me_spare_04 : Bool;
      me_spare_05 : Bool;
      me_spare_06 : Bool;
      me_spare_07 : Bool;
      me_spare_08 : Bool;
      me_spare_09 : Bool;
      me_spare_10 : Bool;   // dipping
      di_new_seed : Bool;   // alter oder neuer Impfling (0=alt/1=neu)
      di_shield_dn : Bool;   // Trichter ist unten
      di_spare_03 : Bool;
      di_spare_04 : Bool;
      di_spare_05 : Bool;
      di_spare_06 : Bool;
      di_spare_07 : Bool;
      di_spare_08 : Bool;
      di_spare_09 : Bool;
      di_spare_10 : Bool;   // neck
      ne_spare_01 : Bool;
      ne_spare_02 : Bool;
      ne_spare_03 : Bool;
      ne_spare_04 : Bool;
      ne_spare_05 : Bool;
      ne_spare_06 : Bool;
      ne_spare_07 : Bool;
      ne_spare_08 : Bool;
      ne_spare_09 : Bool;
      ne_spare_10 : Bool;   // shoulder
      sh_spare_01 : Bool;
      sh_spare_02 : Bool;
      sh_spare_03 : Bool;
      sh_spare_04 : Bool;
      sh_spare_05 : Bool;
      sh_spare_06 : Bool;
      sh_spare_07 : Bool;
      sh_spare_08 : Bool;
      sh_spare_09 : Bool;
      sh_spare_10 : Bool;   // body
      by_spare_01 : Bool;
      by_spare_02 : Bool;
      by_spare_03 : Bool;
      by_spare_04 : Bool;
      by_spare_05 : Bool;
      by_spare_06 : Bool;
      by_spare_07 : Bool;
      by_spare_08 : Bool;
      by_spare_09 : Bool;
      by_spare_10 : Bool;   // endcone
      ec_spare_01 : Bool;
      ec_spare_02 : Bool;
      ec_spare_03 : Bool;
      ec_spare_04 : Bool;
      ec_spare_05 : Bool;
      ec_spare_06 : Bool;
      ec_spare_07 : Bool;
      ec_spare_08 : Bool;
      ec_spare_09 : Bool;
      ec_spare_10 : Bool;   // shut down
      sd_spare_01 : Bool;
      sd_spare_02 : Bool;
      sd_spare_03 : Bool;
      sd_spare_04 : Bool;
      sd_spare_05 : Bool;
      sd_spare_06 : Bool;
      sd_spare_07 : Bool;
      sd_spare_08 : Bool;
      sd_spare_09 : Bool;
      sd_spare_10 : Bool;   // removal
      re_active : Bool;   // Entnahme wurde ausgef黨rt
      re_spare_02 : Bool;
      re_spare_03 : Bool;
      re_spare_04 : Bool;
      re_spare_05 : Bool;
      re_spare_06 : Bool;
      re_spare_07 : Bool;
      re_spare_08 : Bool;
      re_spare_09 : Bool;
      re_spare_10 : Bool;   // melting back
      mb_spare_01 : Bool;
      mb_spare_02 : Bool;
      mb_spare_03 : Bool;
      mb_spare_04 : Bool;
      mb_spare_05 : Bool;
      mb_spare_06 : Bool;
      mb_spare_07 : Bool;
      mb_spare_08 : Bool;
      mb_spare_09 : Bool;
      mb_spare_10 : Bool;   // interne Speicherbits
      pd_sps_spare_01 : Bool;
      pd_sps_spare_02 : Bool;
      pd_sps_spare_03 : Bool;
      pd_sps_spare_04 : Bool;
      pd_sps_spare_05 : Bool;
      pd_sps_spare_06 : Bool;
      pd_sps_spare_07 : Bool;
      pd_sps_spare_08 : Bool;
      pd_sps_spare_09 : Bool;
      pd_sps_spare_10 : Bool;
      me_sps_spare_01 : Bool;
      me_sps_spare_02 : Bool;
      me_sps_spare_03 : Bool;
      me_sps_spare_04 : Bool;
      me_sps_spare_05 : Bool;
      me_sps_spare_06 : Bool;
      me_sps_spare_07 : Bool;
      me_sps_spare_08 : Bool;
      me_sps_spare_09 : Bool;
      me_sps_spare_10 : Bool;
      di_init_melt_temp : Bool;   // speichern Anfangs-Schmelzbadtemp. ausgef黨rt
      di_time_until_dip : Bool;   // speichern der Zeit bis Impfling in Schmelze ausgef黨rt
      di_sps_spare_03 : Bool;
      di_sps_spare_04 : Bool;
      di_sps_spare_05 : Bool;
      di_sps_spare_06 : Bool;
      di_sps_spare_07 : Bool;
      di_sps_spare_08 : Bool;
      di_sps_spare_09 : Bool;
      di_sps_spare_10 : Bool;
      ne_init_xt_pos : Bool;   // speichern Anfangs-Kristallpos. ausgef黨rt
      ne_init_cr_pos : Bool;   // speichern Anfangs-Tiegelposition ausgef黨rt
      ne_init_melt_temp : Bool;   // speichern Anfangs-Schmelzbadtemp. ausgef黨rt
      ne_low_temp_inc : Bool;   // speichern niedrigstes Temp.Inkrement ausgef黨rt
      ne_init_htr_temp : Bool;   // speichern Heizertemp
      ne_sps_spare_06 : Bool;
      ne_sps_spare_07 : Bool;
      ne_sps_spare_08 : Bool;
      ne_sps_spare_09 : Bool;
      ne_sps_spare_10 : Bool;
      sh_start_dia : Bool;   // speichern Startdurchmesser ausgef黨rt
      sh_init_htr_temp : Bool;   // speichern Heizertemp
      sh_sps_spare_03 : Bool;
      sh_sps_spare_04 : Bool;
      sh_sps_spare_05 : Bool;
      sh_sps_spare_06 : Bool;
      sh_sps_spare_07 : Bool;
      sh_sps_spare_08 : Bool;
      sh_sps_spare_09 : Bool;
      sh_sps_spare_10 : Bool;
      by_low_temp_inc : Bool;   // speichern niedrigstes Temp.Inkrement ausgef黨rt
      by_first_dia : Bool;   // speichern Startdurchmesser ausgef黨rt
      by_init_htr_temp : Bool;   // speichern Heizertemp
      by_sps_spare_04 : Bool;
      by_sps_spare_05 : Bool;
      by_sps_spare_06 : Bool;
      by_sps_spare_07 : Bool;
      by_sps_spare_08 : Bool;
      by_sps_spare_09 : Bool;
      by_sps_spare_10 : Bool;
      ec_init_htr_temp : Bool;   // speichern Heizertemp
      ec_sps_spare_02 : Bool;
      ec_sps_spare_03 : Bool;
      ec_sps_spare_04 : Bool;
      ec_sps_spare_05 : Bool;
      ec_sps_spare_06 : Bool;
      ec_sps_spare_07 : Bool;
      ec_sps_spare_08 : Bool;
      ec_sps_spare_09 : Bool;
      ec_sps_spare_10 : Bool;
      sd_sps_spare_01 : Bool;
      sd_sps_spare_02 : Bool;
      sd_sps_spare_03 : Bool;
      sd_sps_spare_04 : Bool;
      sd_sps_spare_05 : Bool;
      sd_sps_spare_06 : Bool;
      sd_sps_spare_07 : Bool;
      sd_sps_spare_08 : Bool;
      sd_sps_spare_09 : Bool;
      sd_sps_spare_10 : Bool;
      re_next_cr_pos : Bool;   // speichern Tiegelposition f黵 n鋍hstes Ankeimen ausgef黨rt
      re_sps_spare_02 : Bool;
      re_sps_spare_03 : Bool;
      re_sps_spare_04 : Bool;
      re_sps_spare_05 : Bool;
      re_sps_spare_06 : Bool;
      re_sps_spare_07 : Bool;
      re_sps_spare_08 : Bool;
      re_sps_spare_09 : Bool;
      re_sps_spare_10 : Bool;
      mb_sps_spare_01 : Bool;
      mb_sps_spare_02 : Bool;
      mb_sps_spare_03 : Bool;
      mb_sps_spare_04 : Bool;
      mb_sps_spare_05 : Bool;
      mb_sps_spare_06 : Bool;
      mb_sps_spare_07 : Bool;
      mb_sps_spare_08 : Bool;
      mb_sps_spare_09 : Bool;
      mb_sps_spare_10 : Bool;
   END_VAR
BEGIN
END_DATA_BLOCK

DATA_BLOCK "BM_GRW_REC_DINT"   // DB702
{ S7_Optimized_Access := 'FALSE' }
VERSION : 0.0
// --------------------------------------------------------------------------------
// program     :        GRW_REC_DINT
// description :        dint data for growth record
// name        :        mb
// date        :        27.11.09
// --------------------------------------------------------------------------------
   VAR
      elapsed_time : DInt;   // gesamte Prozesszeit
      phase_spare_02 : DInt;
      phase_spare_03 : DInt;
      phase_spare_04 : DInt;
      phase_spare_05 : DInt;
      phase_spare_06 : DInt;
      phase_spare_07 : DInt;
      phase_spare_08 : DInt;
      phase_spare_09 : DInt;
      phase_spare_10 : DInt;
      pd_elapsed_time : DInt;   // insgesamt vergangene Prozesszeit
      pd_phase_time : DInt;   // aktuelle/letzte Phasendauer
      pd_to_min_prs : DInt;   // Zeit bis Enddruck erreicht
      pd_retry : DInt;
      pd_spare_05 : DInt;
      pd_spare_06 : DInt;
      pd_spare_07 : DInt;
      pd_spare_08 : DInt;
      pd_spare_09 : DInt;
      pd_spare_10 : DInt;
      me_elapsed_time : DInt;   // insgesamt vergangene Prozesszeit
      me_phase_time : DInt;   // aktuelle/letzte Phasendauer
      me_melt_time : DInt;   // Zeit bis Aufschmelzen beendet
      me_spare_04 : DInt;
      me_spare_05 : DInt;
      me_spare_06 : DInt;
      me_spare_07 : DInt;
      me_spare_08 : DInt;
      me_spare_09 : DInt;
      me_spare_10 : DInt;
      di_elapsed_time : DInt;   // insgesamt vergangene Prozesszeit
      di_phase_time : DInt;   // aktuelle/letzte Phasendauer
      di_shield_dn : DInt;   // Zeit bis Trichter unten
      di_time_until_dip : DInt;   // Zeit bis Impfling in Schmelze
      di_spare_05 : DInt;
      di_spare_06 : DInt;
      di_spare_07 : DInt;
      di_spare_08 : DInt;
      di_spare_09 : DInt;
      di_spare_10 : DInt;
      ne_elapsed_time : DInt;   // insgesamt vergangene Prozesszeit
      ne_phase_time : DInt;   // aktuelle/letzte Phasendauer
      ne_spare_03 : DInt;
      ne_spare_04 : DInt;
      ne_spare_05 : DInt;
      ne_spare_06 : DInt;
      ne_spare_07 : DInt;
      ne_spare_08 : DInt;
      ne_spare_09 : DInt;
      ne_spare_10 : DInt;
      sh_elapsed_time : DInt;   // insgesamt vergangene Prozesszeit
      sh_phase_time : DInt;   // aktuelle/letzte Phasendauer
      sh_spare_03 : DInt;
      sh_spare_04 : DInt;
      sh_spare_05 : DInt;
      sh_spare_06 : DInt;
      sh_spare_07 : DInt;
      sh_spare_08 : DInt;
      sh_spare_09 : DInt;
      sh_spare_10 : DInt;
      by_elapsed_time : DInt;   // insgesamt vergangene Prozesszeit
      by_phase_time : DInt;   // aktuelle/letzte Phasendauer
      by_spare_03 : DInt;
      by_spare_04 : DInt;
      by_spare_05 : DInt;
      by_spare_06 : DInt;
      by_spare_07 : DInt;
      by_spare_08 : DInt;
      by_spare_09 : DInt;
      by_spare_10 : DInt;
      ec_elapsed_time : DInt;   // insgesamt vergangene Prozesszeit
      ec_phase_time : DInt;   // aktuelle/letzte Phasendauer
      ec_spare_03 : DInt;
      ec_spare_04 : DInt;
      ec_spare_05 : DInt;
      ec_spare_06 : DInt;
      ec_spare_07 : DInt;
      ec_spare_08 : DInt;
      ec_spare_09 : DInt;
      ec_spare_10 : DInt;
      sd_elapsed_time : DInt;   // insgesamt vergangene Prozesszeit
      sd_phase_time : DInt;   // aktuelle/letzte Phasendauer
      sd_spare_03 : DInt;
      sd_spare_04 : DInt;
      sd_spare_05 : DInt;
      sd_spare_06 : DInt;
      sd_spare_07 : DInt;
      sd_spare_08 : DInt;
      sd_spare_09 : DInt;
      sd_spare_10 : DInt;
      re_elapsed_time : DInt;   // insgesamt vergangene Prozesszeit
      re_phase_time : DInt;   // aktuelle/letzte Phasendauer
      re_spare_03 : DInt;
      re_spare_04 : DInt;
      re_spare_05 : DInt;
      re_spare_06 : DInt;
      re_spare_07 : DInt;
      re_spare_08 : DInt;
      re_spare_09 : DInt;
      re_spare_10 : DInt;
      mb_elapsed_time : DInt;   // insgesamt vergangene Prozesszeit
      mb_phase_time : DInt;   // aktuelle/letzte Phasendauer
      mb_spare_03 : DInt;
      mb_spare_04 : DInt;
      mb_spare_05 : DInt;
      mb_spare_06 : DInt;
      mb_spare_07 : DInt;
      mb_spare_08 : DInt;
      mb_spare_09 : DInt;
      mb_spare_10 : DInt;
   END_VAR
BEGIN
END_DATA_BLOCK

DATA_BLOCK "BM_GRW_REC_REAL"   // DB703
{ S7_Optimized_Access := 'FALSE' }
VERSION : 0.0
// --------------------------------------------------------------------------------
// program:             GRW_REC_REAL
// description :        REAL data for growth record
// name:                mb
// date        :        23.11.09
// --------------------------------------------------------------------------------
   VAR
      htr_pwr_csp : Real;   // heater power consumption
      ar_gas_csp : Real;   // argon gas consumption
      phase_spare_03 : Real;
      phase_spare_04 : Real;
      phase_spare_05 : Real;
      phase_spare_06 : Real;
      phase_spare_07 : Real;
      phase_spare_08 : Real;
      phase_spare_09 : Real;
      phase_spare_10 : Real;
      phase_spare_11 : Real;
      phase_spare_12 : Real;
      phase_spare_13 : Real;
      phase_spare_14 : Real;
      phase_spare_15 : Real;
      phase_spare_16 : Real;
      phase_spare_17 : Real;
      phase_spare_18 : Real;
      phase_spare_19 : Real;
      phase_spare_20 : Real;
      phase_spare_21 : Real;
      phase_spare_22 : Real;
      phase_spare_23 : Real;
      phase_spare_24 : Real;
      phase_spare_25 : Real;
      phase_spare_26 : Real;
      phase_spare_27 : Real;
      phase_spare_28 : Real;
      phase_spare_29 : Real;
      phase_spare_30 : Real;
      phase_spare_31 : Real;
      phase_spare_32 : Real;
      phase_spare_33 : Real;
      phase_spare_34 : Real;
      phase_spare_35 : Real;
      phase_spare_36 : Real;
      phase_spare_37 : Real;
      phase_spare_38 : Real;
      phase_spare_39 : Real;
      phase_spare_40 : Real;
      pd_final_prs : Real;   // erreichter Enddruck
      pd_leakrate : Real;   // Leckrate
      pd_spare_03 : Real;
      pd_spare_04 : Real;
      pd_spare_05 : Real;
      pd_spare_06 : Real;
      pd_spare_07 : Real;
      pd_spare_08 : Real;
      pd_spare_09 : Real;
      pd_spare_10 : Real;
      pd_spare_11 : Real;
      pd_spare_12 : Real;
      pd_spare_13 : Real;
      pd_spare_14 : Real;
      pd_spare_15 : Real;
      pd_spare_16 : Real;
      pd_spare_17 : Real;
      pd_spare_18 : Real;
      pd_spare_19 : Real;
      pd_spare_20 : Real;
      pd_spare_21 : Real;
      pd_spare_22 : Real;
      pd_spare_23 : Real;
      pd_spare_24 : Real;
      pd_spare_25 : Real;
      pd_spare_26 : Real;
      pd_spare_27 : Real;
      pd_spare_28 : Real;
      pd_spare_29 : Real;
      pd_spare_30 : Real;
      pd_spare_31 : Real;
      pd_spare_32 : Real;
      pd_spare_33 : Real;
      pd_spare_34 : Real;
      pd_spare_35 : Real;
      pd_spare_36 : Real;
      pd_spare_37 : Real;
      pd_spare_38 : Real;
      pd_spare_39 : Real;
      pd_spare_40 : Real;
      me_spare_01 : Real;
      me_spare_02 : Real;
      me_spare_03 : Real;
      me_spare_04 : Real;
      me_spare_05 : Real;
      me_spare_06 : Real;
      me_spare_07 : Real;
      me_spare_08 : Real;
      me_spare_09 : Real;
      me_spare_10 : Real;
      me_spare_11 : Real;
      me_spare_12 : Real;
      me_spare_13 : Real;
      me_spare_14 : Real;
      me_spare_15 : Real;
      me_spare_16 : Real;
      me_spare_17 : Real;
      me_spare_18 : Real;
      me_spare_19 : Real;
      me_spare_20 : Real;
      me_spare_21 : Real;
      me_spare_22 : Real;
      me_spare_23 : Real;
      me_spare_24 : Real;
      me_spare_25 : Real;
      me_spare_26 : Real;
      me_spare_27 : Real;
      me_spare_28 : Real;
      me_spare_29 : Real;
      me_spare_30 : Real;
      me_spare_31 : Real;
      me_spare_32 : Real;
      me_spare_33 : Real;
      me_spare_34 : Real;
      me_spare_35 : Real;
      me_spare_36 : Real;
      me_spare_37 : Real;
      me_spare_38 : Real;
      me_spare_39 : Real;
      me_spare_40 : Real;
      di_init_melt_temp : Real;   // Anfangs-Schmelzbadtemp.
      di_final_htr_1_pwr : Real;   // Heizer 1 Leistung am Phasenende
      di_spare_03 : Real;
      di_spare_04 : Real;
      di_spare_05 : Real;
      di_spare_06 : Real;
      di_spare_07 : Real;
      di_spare_08 : Real;
      di_spare_09 : Real;
      di_spare_10 : Real;
      di_spare_11 : Real;
      di_spare_12 : Real;
      di_spare_13 : Real;
      di_spare_14 : Real;
      di_spare_15 : Real;
      di_spare_16 : Real;
      di_spare_17 : Real;
      di_spare_18 : Real;
      di_spare_19 : Real;
      di_spare_20 : Real;
      di_spare_21 : Real;
      di_spare_22 : Real;
      di_spare_23 : Real;
      di_spare_24 : Real;
      di_spare_25 : Real;
      di_spare_26 : Real;
      di_spare_27 : Real;
      di_spare_28 : Real;
      di_spare_29 : Real;
      di_spare_30 : Real;
      di_spare_31 : Real;
      di_spare_32 : Real;
      di_spare_33 : Real;
      di_spare_34 : Real;
      di_spare_35 : Real;
      di_spare_36 : Real;
      di_spare_37 : Real;
      di_spare_38 : Real;
      di_spare_39 : Real;
      di_spare_40 : Real;
      ne_init_cr_pos : Real;   // Anfangs-Tiegelpos.
      ne_init_melt_temp : Real;   // Anfangs-Schmelzbadtemp.
      ne_final_melt_temp : Real;   // finale-Schmelzbadtemp.
      ne_low_temp_inc : Real;   // niedrigstes Temp.Inc.
      ne_final_temp_inc : Real;   // finales Temp.Inc.
      ne_phase_avg_spd : Real;   // Durchschnittl. Ziehgeschwindigkeit (gesamte Halsl鋘ge)
      ne_final_avg_spd : Real;   // finale Durchschnittl. Ziehgeschwindigkeit
      ne_final_htr_1_pwr : Real;   // Heizer 1 Leistung am Phasenende
      ne_spare_09 : Real;
      ne_spare_10 : Real;
      ne_spare_11 : Real;
      ne_spare_12 : Real;
      ne_spare_13 : Real;
      ne_spare_14 : Real;
      ne_spare_15 : Real;
      ne_spare_16 : Real;
      ne_spare_17 : Real;
      ne_spare_18 : Real;
      ne_spare_19 : Real;
      ne_spare_20 : Real;
      ne_spare_21 : Real;
      ne_spare_22 : Real;
      ne_spare_23 : Real;
      ne_spare_24 : Real;
      ne_spare_25 : Real;
      ne_spare_26 : Real;
      ne_spare_27 : Real;
      ne_spare_28 : Real;
      ne_spare_29 : Real;
      ne_spare_30 : Real;
      ne_spare_31 : Real;
      ne_spare_32 : Real;
      ne_spare_33 : Real;
      ne_spare_34 : Real;
      ne_spare_35 : Real;
      ne_spare_36 : Real;
      ne_spare_37 : Real;
      ne_spare_38 : Real;
      ne_spare_39 : Real;
      ne_spare_40 : Real;
      sh_phase_avg_grth : Real;   // Durchschnittl. Wachstumsgeschwindigkeit (gesamte Schulter)
      sh_final_temp_inc : Real;   // finales Temp.Inc.
      sh_weight : Real;   // Gewicht der Schulter
      sh_final_htr_1_pwr : Real;   // Heizer 1 Leistung am Phasenende
      sh_spare_05 : Real;
      sh_spare_06 : Real;
      sh_spare_07 : Real;
      sh_spare_08 : Real;
      sh_spare_09 : Real;
      sh_spare_10 : Real;
      sh_spare_11 : Real;
      sh_spare_12 : Real;
      sh_spare_13 : Real;
      sh_spare_14 : Real;
      sh_spare_15 : Real;
      sh_spare_16 : Real;
      sh_spare_17 : Real;
      sh_spare_18 : Real;
      sh_spare_19 : Real;
      sh_spare_20 : Real;
      sh_spare_21 : Real;
      sh_spare_22 : Real;
      sh_spare_23 : Real;
      sh_spare_24 : Real;
      sh_spare_25 : Real;
      sh_spare_26 : Real;
      sh_spare_27 : Real;
      sh_spare_28 : Real;
      sh_spare_29 : Real;
      sh_spare_30 : Real;
      sh_spare_31 : Real;
      sh_spare_32 : Real;
      sh_spare_33 : Real;
      sh_spare_34 : Real;
      sh_spare_35 : Real;
      sh_spare_36 : Real;
      sh_spare_37 : Real;
      sh_spare_38 : Real;
      sh_spare_39 : Real;
      sh_spare_40 : Real;
      by_phase_avg_spd : Real;   // Durchschnittl. Ziehgeschwindigkeit (gesamt)
      by_final_avg_spd : Real;   // finale Durchschnittl. Ziehgeschwindigkeit
      by_low_temp_inc : Real;   // niedrigstes Temp.Inc.
      by_final_temp_inc : Real;   // finales Temp.Inc.
      by_avg_dia : Real;   // Durchschnittl. Durchmesser
      by_weight : Real;   // Gewicht vom Stab
      by_lenght : Real;   // Stabl鋘ge
      by_total_length : Real;   // Gesamtl鋘ge
      by_rem_cr_wgt : Real;   // verbleibende Siliziummenge im Tiegel
      by_final_cr_pos : Real;   // finale Tiegelpos.
      by_final_htr_1_pwr : Real;   // Heizer 1 Leistung am Phasenende
      by_spare_12 : Real;
      by_spare_13 : Real;
      by_spare_14 : Real;
      by_spare_15 : Real;
      by_spare_16 : Real;
      by_spare_17 : Real;
      by_spare_18 : Real;
      by_spare_19 : Real;
      by_spare_20 : Real;
      by_spare_21 : Real;
      by_spare_22 : Real;
      by_spare_23 : Real;
      by_spare_24 : Real;
      by_spare_25 : Real;
      by_spare_26 : Real;
      by_spare_27 : Real;
      by_spare_28 : Real;
      by_spare_29 : Real;
      by_spare_30 : Real;
      by_spare_31 : Real;
      by_spare_32 : Real;
      by_spare_33 : Real;
      by_spare_34 : Real;
      by_spare_35 : Real;
      by_spare_36 : Real;
      by_spare_37 : Real;
      by_spare_38 : Real;
      by_spare_39 : Real;
      by_spare_40 : Real;
      ec_phase_avg_spd : Real;   // Durchschnittl. Ziehgeschwindigkeit (gesamt)
      ec_final_temp_inc : Real;   // finales Temp.Inc.
      ec_weight : Real;   // Gewicht vom Endkonus
      ec_rem_cr_wgt : Real;   // verbleibende Siliziummenge im Tiegel
      ec_final_htr_1_pwr : Real;   // Heizer 1 Leistung am Phasenende
      ec_spare_06 : Real;
      ec_spare_07 : Real;
      ec_spare_08 : Real;
      ec_spare_09 : Real;
      ec_spare_10 : Real;
      ec_spare_11 : Real;
      ec_spare_12 : Real;
      ec_spare_13 : Real;
      ec_spare_14 : Real;
      ec_spare_15 : Real;
      ec_spare_16 : Real;
      ec_spare_17 : Real;
      ec_spare_18 : Real;
      ec_spare_19 : Real;
      ec_spare_20 : Real;
      ec_spare_21 : Real;
      ec_spare_22 : Real;
      ec_spare_23 : Real;
      ec_spare_24 : Real;
      ec_spare_25 : Real;
      ec_spare_26 : Real;
      ec_spare_27 : Real;
      ec_spare_28 : Real;
      ec_spare_29 : Real;
      ec_spare_30 : Real;
      ec_spare_31 : Real;
      ec_spare_32 : Real;
      ec_spare_33 : Real;
      ec_spare_34 : Real;
      ec_spare_35 : Real;
      ec_spare_36 : Real;
      ec_spare_37 : Real;
      ec_spare_38 : Real;
      ec_spare_39 : Real;
      ec_spare_40 : Real;
      sd_spare_01 : Real;
      sd_spare_02 : Real;
      sd_spare_03 : Real;
      sd_spare_04 : Real;
      sd_spare_05 : Real;
      sd_spare_06 : Real;
      sd_spare_07 : Real;
      sd_spare_08 : Real;
      sd_spare_09 : Real;
      sd_spare_10 : Real;
      sd_spare_11 : Real;
      sd_spare_12 : Real;
      sd_spare_13 : Real;
      sd_spare_14 : Real;
      sd_spare_15 : Real;
      sd_spare_16 : Real;
      sd_spare_17 : Real;
      sd_spare_18 : Real;
      sd_spare_19 : Real;
      sd_spare_20 : Real;
      sd_spare_21 : Real;
      sd_spare_22 : Real;
      sd_spare_23 : Real;
      sd_spare_24 : Real;
      sd_spare_25 : Real;
      sd_spare_26 : Real;
      sd_spare_27 : Real;
      sd_spare_28 : Real;
      sd_spare_29 : Real;
      sd_spare_30 : Real;
      sd_spare_31 : Real;
      sd_spare_32 : Real;
      sd_spare_33 : Real;
      sd_spare_34 : Real;
      sd_spare_35 : Real;
      sd_spare_36 : Real;
      sd_spare_37 : Real;
      sd_spare_38 : Real;
      sd_spare_39 : Real;
      sd_spare_40 : Real;
      re_next_cr_pos : Real;   // n鋍hste Tiegelpos.
      re_final_htr_1_pwr : Real;   // Heizer 1 Leistung am Phasenende
      re_spare_03 : Real;
      re_spare_04 : Real;
      re_spare_05 : Real;
      re_spare_06 : Real;
      re_spare_07 : Real;
      re_spare_08 : Real;
      re_spare_09 : Real;
      re_spare_10 : Real;
      re_spare_11 : Real;
      re_spare_12 : Real;
      re_spare_13 : Real;
      re_spare_14 : Real;
      re_spare_15 : Real;
      re_spare_16 : Real;
      re_spare_17 : Real;
      re_spare_18 : Real;
      re_spare_19 : Real;
      re_spare_20 : Real;
      re_spare_21 : Real;
      re_spare_22 : Real;
      re_spare_23 : Real;
      re_spare_24 : Real;
      re_spare_25 : Real;
      re_spare_26 : Real;
      re_spare_27 : Real;
      re_spare_28 : Real;
      re_spare_29 : Real;
      re_spare_30 : Real;
      re_spare_31 : Real;
      re_spare_32 : Real;
      re_spare_33 : Real;
      re_spare_34 : Real;
      re_spare_35 : Real;
      re_spare_36 : Real;
      re_spare_37 : Real;
      re_spare_38 : Real;
      re_spare_39 : Real;
      re_spare_40 : Real;
      mb_phase_avg_spd : Real;
      mb_final_cr_pos : Real;
      mb_spare_03 : Real;
      mb_spare_04 : Real;
      mb_spare_05 : Real;
      mb_spare_06 : Real;
      mb_spare_07 : Real;
      mb_spare_08 : Real;
      mb_spare_09 : Real;
      mb_spare_10 : Real;
      mb_spare_11 : Real;
      mb_spare_12 : Real;
      mb_spare_13 : Real;
      mb_spare_14 : Real;
      mb_spare_15 : Real;
      mb_spare_16 : Real;
      mb_spare_17 : Real;
      mb_spare_18 : Real;
      mb_spare_19 : Real;
      mb_spare_20 : Real;
      mb_spare_21 : Real;
      mb_spare_22 : Real;
      mb_spare_23 : Real;
      mb_spare_24 : Real;
      mb_spare_25 : Real;
      mb_spare_26 : Real;
      mb_spare_27 : Real;
      mb_spare_28 : Real;
      mb_spare_29 : Real;
      mb_spare_30 : Real;
      mb_spare_31 : Real;
      mb_spare_32 : Real;
      mb_spare_33 : Real;
      mb_spare_34 : Real;
      mb_spare_35 : Real;
      mb_spare_36 : Real;
      mb_spare_37 : Real;
      mb_spare_38 : Real;
      mb_spare_39 : Real;
      mb_spare_40 : Real;   // interne Speicherwerte
      pd_sps_spare_01 : Real;
      pd_sps_spare_02 : Real;
      pd_sps_spare_03 : Real;
      pd_sps_spare_04 : Real;
      pd_sps_spare_05 : Real;
      pd_sps_spare_06 : Real;
      pd_sps_spare_07 : Real;
      pd_sps_spare_08 : Real;
      pd_sps_spare_09 : Real;
      pd_sps_spare_10 : Real;
      me_sps_spare_01 : Real;
      me_sps_spare_02 : Real;
      me_sps_spare_03 : Real;
      me_sps_spare_04 : Real;
      me_sps_spare_05 : Real;
      me_sps_spare_06 : Real;
      me_sps_spare_07 : Real;
      me_sps_spare_08 : Real;
      me_sps_spare_09 : Real;
      me_sps_spare_10 : Real;
      di_sps_spare_01 : Real;
      di_sps_spare_02 : Real;
      di_sps_spare_03 : Real;
      di_sps_spare_04 : Real;
      di_sps_spare_05 : Real;
      di_sps_spare_06 : Real;
      di_sps_spare_07 : Real;
      di_sps_spare_08 : Real;
      di_sps_spare_09 : Real;
      di_sps_spare_10 : Real;
      ne_sps_init_xt_pos : Real;   // Anfangs-Kristallpos.
      ne_sps_init_htr_temp : Real;   // Anfangs-Heizertemp
      ne_sps_spare_03 : Real;
      ne_sps_spare_04 : Real;
      ne_sps_spare_05 : Real;
      ne_sps_spare_06 : Real;
      ne_sps_spare_07 : Real;
      ne_sps_spare_08 : Real;
      ne_sps_spare_09 : Real;
      ne_sps_spare_10 : Real;
      sh_sps_start_dia : Real;   // Startdurchnesser (nur Speicher f黵 Berechnung)
      sh_sps_init_htr_temp : Real;   // Anfangs-Heizertemp
      sh_sps_spare_03 : Real;
      sh_sps_spare_04 : Real;
      sh_sps_spare_05 : Real;
      sh_sps_spare_06 : Real;
      sh_sps_spare_07 : Real;
      sh_sps_spare_08 : Real;
      sh_sps_spare_09 : Real;
      sh_sps_spare_10 : Real;
      by_first_dia : Real;   // Startdurchmesser (nur Speicher f黵 Berechnung)
      by_start_wgt : Real;   // Startgewicht (nur Speicher f黵 Berechnung)
      by_sps_init_htr_temp : Real;   // Anfangs-Heizertemp
      by_sps_spare_04 : Real;
      by_sps_spare_05 : Real;
      by_sps_spare_06 : Real;
      by_sps_spare_07 : Real;
      by_sps_spare_08 : Real;
      by_sps_spare_09 : Real;
      by_sps_spare_10 : Real;
      ec_sps_init_htr_temp : Real;   // Anfangs-Heizertemp
      ec_sps_spare_02 : Real;
      ec_sps_spare_03 : Real;
      ec_sps_spare_04 : Real;
      ec_sps_spare_05 : Real;
      ec_sps_spare_06 : Real;
      ec_sps_spare_07 : Real;
      ec_sps_spare_08 : Real;
      ec_sps_spare_09 : Real;
      ec_sps_spare_10 : Real;
      sd_sps_spare_01 : Real;
      sd_sps_spare_02 : Real;
      sd_sps_spare_03 : Real;
      sd_sps_spare_04 : Real;
      sd_sps_spare_05 : Real;
      sd_sps_spare_06 : Real;
      sd_sps_spare_07 : Real;
      sd_sps_spare_08 : Real;
      sd_sps_spare_09 : Real;
      sd_sps_spare_10 : Real;
      re_sps_rem_si_wgt : Real;
      re_sps_spare_02 : Real;
      re_sps_spare_03 : Real;
      re_sps_spare_04 : Real;
      re_sps_spare_05 : Real;
      re_sps_spare_06 : Real;
      re_sps_spare_07 : Real;
      re_sps_spare_08 : Real;
      re_sps_spare_09 : Real;
      re_sps_spare_10 : Real;
      mb_sps_spare_01 : Real;
      mb_sps_spare_02 : Real;
      mb_sps_spare_03 : Real;
      mb_sps_spare_04 : Real;
      mb_sps_spare_05 : Real;
      mb_sps_spare_06 : Real;
      mb_sps_spare_07 : Real;
      mb_sps_spare_08 : Real;
      mb_sps_spare_09 : Real;
      mb_sps_spare_10 : Real;
   END_VAR
BEGIN
END_DATA_BLOCK

FUNCTION "FLT_BLKMOV" : Void   // FC3, STL
TITLE = Coppy all fault bits into data of CDP
{ S7_Optimized_Access := 'FALSE' }
VERSION : 0.1
   VAR_TEMP
      RETVAL : Int;
   END_VAR
BEGIN

REGION Network 1
         CALL  BLKMOV
         ( SRCBLK  := P#DB142.DBX0.0 BYTE 68,
           RET_VAL := #RETVAL,
           DSTBLK  := P#DB636.DBX0.0 BYTE 68
         );
END_REGION
END_FUNCTION

FUNCTION "CALL_PN_DIAG" : Void   // FC99, STL
TITLE = Call SFC 51 (RDSYSST) used for Profinet Diagnosis
{ S7_Optimized_Access := 'FALSE' }
AUTHOR : ge
VERSION : 0.1
// SZL_ID: W#16#0694:
// Diagnosezustand der Erweiterungsger鋞e im zentralen Aufbau / 
// der Stationen eines IO-Controllersystems
// Status-Bit = 1: mind. eine Baugruppe 
// des Rack/Station ist gest鰎t oder deaktiviert)
// 
// Index: 100-115: Dezentrale Baugruppe am PROFINET IO
BEGIN

REGION Network 1
         CALL  RDSYSST
         ( REQ        := TRUE,
           SZL_ID     := WORD#16#0694,
           INDEX      := WORD#16#0064,  //IO-Sytemnumber: dez: 100 >>hex 64
           RET_VAL    := %DB1000.DBW272,
           BUSY       := %DB1000.DBX274.0,
           SZL_HEADER := P#DB1000.DBX286.0 BYTE 4,
           DR         := P#DB1000.DBX0.0 BYTE 258
         );
END_REGION
END_FUNCTION

FUNCTION "SysTimeFlag" : Void   // FC110, STL
TITLE = System Timer Flags
{ S7_Optimized_Access := 'FALSE' }
AUTHOR : hp
FAMILY : System
NAME : TmeFlags
VERSION : 1.0
// Project    : Common
// Programmer : hp
// Release    : 04.12.1999
// Function   : Set all time flags for one cycle
// Changes    :
BEGIN

REGION Network 1: set logical 0 / 1
         A     "Tag_1";
         AN    "Tag_1";
         =     "Tag_1";

         O     "Tag_2";
         ON    "Tag_2";
         =     "Tag_2";
END_REGION

REGION Network 2: Reset all time flags
         A     "Tag_2";
         R     "Tag_3";
         R     "Tag_4";
         R     "Tag_5";
         R     "Tag_6";
         R     "Tag_7";
         R     "Tag_8";
         R     "Tag_9";
         R     "Tag_10";
END_REGION

REGION Network 3: Set time flag 100 ms
         A     "Tag_11";
         FP    "Tag_12";  // positive edge 100 ms cycle
         =     "Tag_13";  // impuls 100 ms

         A     "Tag_13";
         S     "Tag_3";  // Set tick for one cycle
END_REGION

REGION Network 4: Set time flag 200 ms
         A     "Tag_14";
         FP    "Tag_15";  // positive edge 200 ms cycle
         =     "Tag_16";  // impuls 200 ms

         A     "Tag_16";
         S     "Tag_4";  // Set tick for one cycle
END_REGION

REGION Network 5: Set time flag 400 ms
         A     "Tag_17";
         FP    "Tag_18";  // positive edge 400 ms cycle
         =     "Tag_19";  // impuls 400 ms

         A     "Tag_19";
         S     "Tag_5";  // Set tick for one cycle
END_REGION

REGION Network 6: Set time flag 500 ms
         A     "Tag_20";
         FP    "Tag_21";  // positive edge 500 ms cycle
         =     "Tag_22";  // impuls 500 ms

         A     "Tag_22";
         S     "Tag_6";  // Set tick for one cycle
END_REGION

REGION Network 7: Set time flag 800 ms
         A     "Tag_23";
         FP    "Tag_24";  // positive edge 800 ms cycle
         =     "Tag_25";  // impuls 800 ms

         A     "Tag_25";
         S     "Tag_7";  // Set tick for one cycle
END_REGION

REGION Network 8: Set time flag 1000 ms
         A     "Tag_26";
         FP    "Tag_27";  // positive edge 1000 ms cycle
         =     "Tag_28";  // impuls 1000 ms

         A     "Tag_28";
         S     "Tag_8";  // Set tick for one cycle
END_REGION

REGION Network 9: Set time flag 1600 ms
         A     "Tag_29";
         FP    "Tag_30";  // positive edge 1600 ms cycle
         =     "Tag_31";  // impuls 1600 ms

         A     "Tag_31";
         S     "Tag_9";  // Set tick for one cycle
END_REGION

REGION Network 10: Set time flag 2000 ms
         A     "Tag_32";
         FP    "Tag_33";  // positive edge 2000 ms cycle
         =     "Tag_34";  // impuls 2000 ms

         A     "Tag_34";
         S     "Tag_10";  // Set tick for one cycle
END_REGION
END_FUNCTION

FUNCTION "SysOndelay" : Bool   // FC111, STL
TITLE = Variable OnDelay
{ S7_Optimized_Access := 'FALSE' }
AUTHOR : HL
FAMILY : System
NAME : OnDelay
VERSION : 1.0
// Project    : Common
// Programmer : BPS (HL)
// Release    : 12.08.1998
// Function   : Variable Ondelay Function
//              Time Base: #Tick (100 ms ... 1000 ms)
//              Max. OnDelay Time = 32767 s
// Changes    :
   VAR_INPUT
      SetTime : Int;   // Setpoint OnDelay Time [s]
      Tick : Bool;   // System Tick
      DIN : Bool;   // Digital Input To Start
   END_VAR
   VAR_IN_OUT
      ActTime : Int;   // Actual Time [s]
   END_VAR
   VAR_TEMP
      DOUT : Bool;   // Digital Output Ondelayed
   END_VAR
BEGIN

REGION Network 1
   // Reset Digital Output:
         A     "Tag_1";
         =     #DOUT;

   // Test Digital Input = 0  -> Reset All Values
         AN    #DIN;
         JC    RSET;

   // Test TickTime Over:
         AN    #Tick;
         JC    TACT;  // =TACT: Test Actual Time

   // Test Delay Time Over:
         L     #ActTime;  // Increment Actual Timer
         L     1;
         +I;
         T     #ActTime;  // Save Actual Time


   TACT: NOP   0;  // TACT: Test Actual OnDelay Time
         L     #ActTime;
         L     #SetTime;
         >=I;  // Test ActTime >= SetTime
         =     #DOUT;  // Set Digital Output
         JC    FIN;  // =FIN
         JU    END;  // =END

   RSET: NOP   0;  // =RSET: Reset All Values
         L     0;
         T     #ActTime;  // Reset Actual Delay Time

   FIN:  NOP   0;  // =FIN:
         T     #ActTime;  // Stop Actual Time If Setpoint Reached

   END:  NOP   0;  // =END:

         A     #DOUT;
         =     #SysOndelay;  //Set Return Value
END_REGION
END_FUNCTION

FUNCTION "SysOffdelay" : Bool   // FC112, STL
TITLE = Variable OffDelay
{ S7_Optimized_Access := 'FALSE' }
AUTHOR : HL
FAMILY : System
NAME : OffDelay
VERSION : 0.0
// Project    : Common
// Programmer : Helmut Lausmann
// Release    : 12.08.1998
// Function   : Variable OffDelay Function
//              Time Base: #Tick (100 ms ... 1000 ms))
//              Max OffDelay Time = 32767 s
// Changes    :
   VAR_INPUT
      SetTime : Int;   // Setpoint OffDelay Time [s]
      Tick : Bool;   // System Tick
      DIN : Bool;   // Digital Input To Start
   END_VAR
   VAR_IN_OUT
      ActTime : Int;   // Actual Time [s]
   END_VAR
   VAR_TEMP
      DOUT : Bool;   // Digital Output Offdelayed
   END_VAR
BEGIN

REGION Network 1
   // Test Digital Input = 1
         A     #DIN;
         =     #DOUT;
         JC    PSET;  // =PSET: Preset Of OffDelay

   // Test Actual Time For Zero
         L     #ActTime;
         L     0;
         ==I;
         AN    #DIN;  // Test Digital Input
         JC    END;  // =REFR:

         AN    #Tick;
         JC    TACT;  // =TACT:
   //
   // Tick Over : Increment Actual Time
         L     #ActTime;  // Increment Actual Time
         L     1;
         +I;
         T     #ActTime;  // Save Actual Time

   // Test Actual OffDelay Time:
   TACT: NOP   0;
         L     #ActTime;
         L     #SetTime;
         <=I;  // Test ActTime <= SetTime
         =     #DOUT;  // Set Digital Output
         JC    END;  // =REFR
         L     0;
         T     #ActTime;  // Reset Actual Counter
         JU    END;  // =REFR:

   PSET: NOP   0;  // PSET: Preset Of OffDelay Counter
         L     1;  // Reset Actual Delay Time
         T     #ActTime;

   //
   END:  NOP   0;  // NEND

         A     #DOUT;
         =     #SysOffdelay;  //Set Return Value
END_REGION
END_FUNCTION